FUNCTION_BLOCK VaccumSlave (* Basic Function Block Type *)
  (* Standard: 61499-2 *)
  (* Version 0.2, 2003-12-04, JHC, Rockwell Automation, Renamed for better indexing. *)
  (* Version 0.1, 2002-11-05, JHC, Rockwell Automation, Corrected missing ST element in Algorithm REQ. *)
  (* Version 0.0, 2000-05-30, JHC, Rockwell Automation *)
  (* Compiler header: package fb.rt.pnp; *)
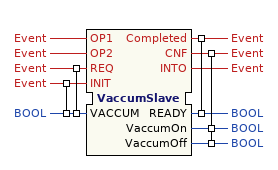
  EVENT_INPUT
    OP1; (* Initialization Request *)
    OP2; (* Normal Execution Request *)
    REQ WITH VACCUM;
    INIT WITH VACCUM;
  END_EVENT
  EVENT_OUTPUT
    Completed WITH READY; (* Initialization Confirm *)
    CNF WITH VaccumOn, VaccumOff;
    INTO;
  END_EVENT
  VAR_INPUT
    VACCUM : BOOL; (* Input event qualifier *)
  END_VAR
  VAR_OUTPUT
    READY : BOOL; (* Output event qualifier *)
    VaccumOn : BOOL; (* Output event qualifier *)
    VaccumOff : BOOL; (* Output event qualifier *)
  END_VAR
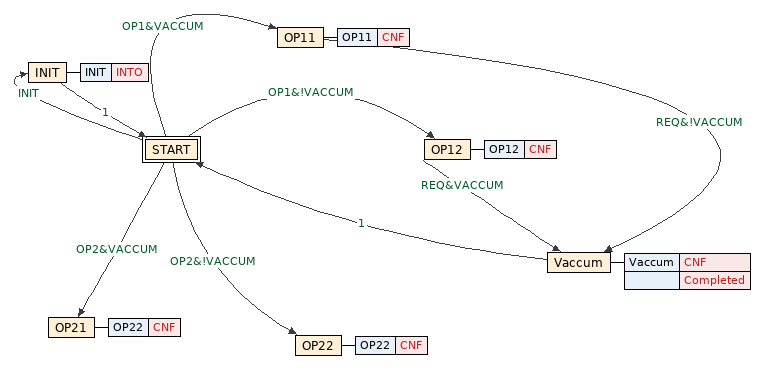
  EC_STATES
    START; (* Initial State *)
    OP11 : OP11 -> CNF; (* Initialization *)
    OP22 : OP22 -> CNF; (* Normal execution *)
    OP12 : OP12 -> CNF; (* Initialization *)
    OP21 : OP22 -> CNF; (* Normal execution *)
    Vaccum : Vaccum -> CNF, -> Completed;
    INIT : INIT -> INTO;
  END_STATES
  EC_TRANSITIONS
    START TO OP11 := OP1&VACCUM;
    START TO OP22 := OP2&!VACCUM;
    START TO OP12 := OP1&!VACCUM;
    START TO OP21 := OP2&VACCUM;
    OP12 TO Vaccum := REQ&VACCUM;
    Vaccum TO START := 1;
    OP11 TO Vaccum := REQ&!VACCUM;
    START TO INIT := INIT;
    INIT TO START := 1;
  END_TRANSITIONS
  ALGORITHM REQ IN ST: (* Normally executed algorithm *)

  END_ALGORITHM
  ALGORITHM OP11 IN ST:
VaccumOff := TRUE;
VaccumOn := FALSE;
READY := FALSE;
System.out.println("OP11!!");
  END_ALGORITHM
  ALGORITHM OP12 IN ST:
VaccumOff := FALSE;
VaccumOn := TRUE;
READY := FALSE;
System.out.println("OP12!!");
  END_ALGORITHM
  ALGORITHM OP21 IN ST:
VaccumOff := TRUE;
VaccumOn := FALSE;
READY := FALSE;
System.out.println("OP21!!");
  END_ALGORITHM
  ALGORITHM OP22 IN ST:
VaccumOff := TRUE;
VaccumOn := FALSE;
READY := FALSE;
System.out.println("OP22!!");
  END_ALGORITHM
  ALGORITHM Vaccum IN ST:
READY := TRUE;
System.out.println("Vaccum!!");
  END_ALGORITHM
  ALGORITHM INIT IN ST:
VACCUM := FALSE;
  END_ALGORITHM
END_FUNCTION_BLOCK
